PROGRAM PRG_IpcControllerMain
VAR
END_VAR
VAR
    fbLocalTime     : FB_LocalSystemTime;  // Synchronizes with Windows clock
    dtCurrentTime   : DT;
	fbVisControl	: FB_VisControl;
END_VAR

fbVisControl();
// GET LOCAL TIME - First call start
fbLocalTime( 
    bEnable := TRUE,        // trigger initial sync
    dwCycle := 60           // resync every 60 s
);

// After first sync, FB bValid becomes TRUE
IF fbLocalTime.bValid THEN
// Update dtCurrentTime each cycle
    dtCurrentTime := SYSTEMTIME_TO_DT(fbLocalTime.systemTime);
END_IF

GVL_Controller.dtSystemTime := dtCurrentTime;

END_PROGRAM

(* stored: Version 1.1.0.1
   POU PRG_IpcControllerMain: Id {075ea502-c30b-43b0-8467-21d133ac9e69}, SpecialFunc None *)
